{attribute 'GeneratedUsingTerminal: EL3413-0000-0016'}
{attribute addProperty BoxType "EL3413-0000-0016"}
{attribute addProperty Id "STATUSAT %I*STATUS_1538B4EA8CurrentAT %I*DINT4VoltageAT %I*DINT4Active_powerAT %I*DINT4IndexAT %I*USINT1Variant_valueAT %I*DINT4"}
{attribute addProperty CRC "878620244"}
{attribute addProperty Size "25"}
TYPE PM_Inputs_Channel_345EAE54 :
STRUCT
	{attribute addProperty Name "STATUS"}
	STATUS AT %I* : STATUS_1538B4EA;
	{attribute addProperty Name "Current"}
	Current AT %I* : DINT;
	{attribute addProperty Name "Voltage"}
	Voltage AT %I* : DINT;
	{attribute addProperty Name "Active_power"}
	Active_power AT %I* : DINT;
	{attribute addProperty Name "Index"}
	Index AT %I* : USINT;
	{attribute addProperty Name "Variant_value"}
	Variant_value AT %I* : DINT;
END_STRUCT
END_TYPE

(* stored: Version 1.2.0.0, ProductVersion 3.1.4024.9
   DUT PM_Inputs_Channel_345EAE54: Id {542d0e27-68f0-42d4-92f2-0ced72034b7f} *)
